// TIA Portal V18 export
FUNCTION "Block_LD" : Void   // FC2, LAD
{ S7_Optimized_Access := 'TRUE' }
// stored: SetENOAutomatically false
   VAR_TEMP
      "A" : Bool;
      "B" : Bool;
      C : Bool;
      D : Bool;
      QU : Bool;
      QD : Bool;
      PT : Time;
      ET : Time;
      PV : Int;
      CV : Int;
   END_VAR
BEGIN

REGION Network 1
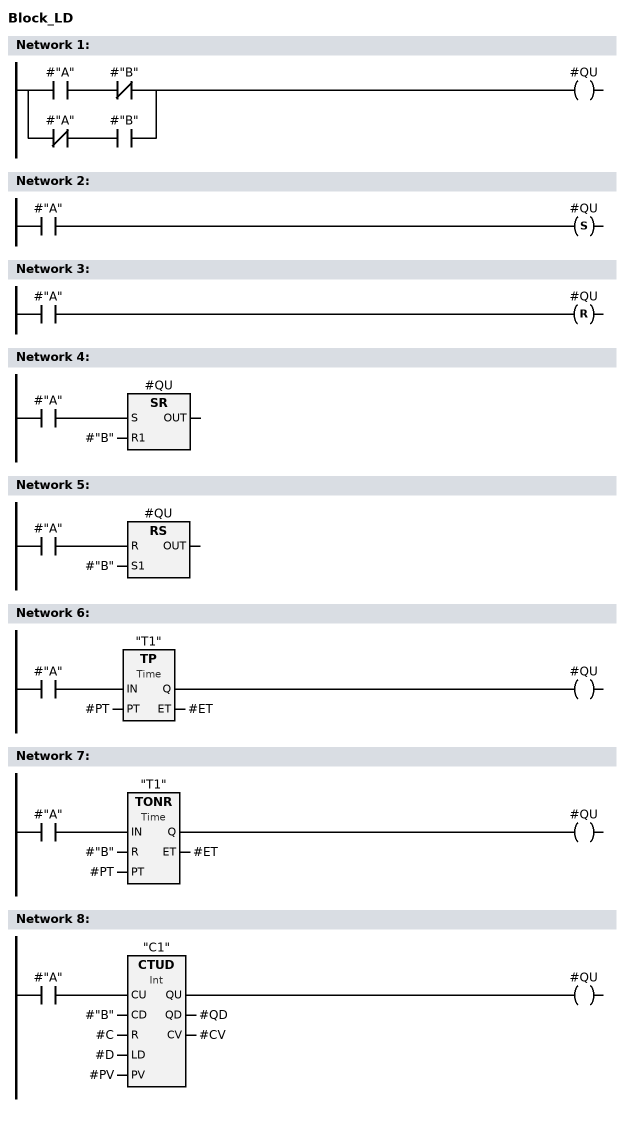
   RUNG wire#powerrail
      Contact( #"A" )
      I_Contact( #"B" )
      wire#w1
      Coil( #QU )
   END_RUNG
   RUNG wire#powerrail
      I_Contact( #"A" )
      Contact( #"B" )
   END_RUNG wire#w1
   // the same network as SCL:
   #QU := (#"A" AND NOT #"B") OR (NOT #"A" AND #"B");
END_REGION

REGION Network 2
   RUNG wire#powerrail
      Contact( #"A" )
      S_Coil( #QU )
   END_RUNG
   // the same network as SCL:
   IF #"A" THEN #QU := TRUE; END_IF;
END_REGION

REGION Network 3
   RUNG wire#powerrail
      Contact( #"A" )
      R_Coil( #QU )
   END_RUNG
   // the same network as SCL:
   IF #"A" THEN #QU := FALSE; END_IF;
END_REGION

REGION Network 4
   RUNG wire#powerrail
      Contact( #"A" )
      S_SR(operand := #QU, r1 := #"B")
   END_RUNG
   // the same network as SCL:
   IF #"A" THEN
       #QU := TRUE;   // SR flip-flop
   END_IF;
   IF #"B" THEN #QU := FALSE; END_IF;
END_REGION

REGION Network 5
   RUNG wire#powerrail
      Contact( #"A" )
      S_RS(operand := #QU, s1 := #"B")
   END_RUNG
   // the same network as SCL:
   IF #"A" THEN
       #QU := FALSE;   // RS flip-flop
   END_IF;
   IF #"B" THEN #QU := TRUE; END_IF;
END_REGION

REGION Network 6
   RUNG wire#powerrail
      Contact( #"A" )
      { S7_Templates := "time_type := Time" } "T1".TP(pt := #PT, et => #ET)
      Coil( #QU )
   END_RUNG
   // the same network as SCL:
   "T1".TP(IN := #"A", PT := #PT, ET => #ET);
   #QU := "T1".Q;
END_REGION

REGION Network 7
   RUNG wire#powerrail
      Contact( #"A" )
      { S7_Templates := "time_type := Time" } "T1".TONR(r := #"B", pt := #PT, et => #ET)
      Coil( #QU )
   END_RUNG
   // the same network as SCL:
   "T1".TONR(IN := #"A", R := #"B", PT := #PT, ET => #ET);
   #QU := "T1".Q;
END_REGION

REGION Network 8
   RUNG wire#powerrail
      Contact( #"A" )
      { S7_Templates := "value_type := Int" } "C1".CTUD(cd := #"B", r := #C, ld := #D, pv := #PV, qd => #QD, cv => #CV)
      Coil( #QU )
   END_RUNG
   // the same network as SCL:
   "C1".CTUD(CU := #"A", CD := #"B", R := #C, LD := #D, PV := #PV, QD => #QD, CV => #CV);
   #QU := "C1".QU;
END_REGION
END_FUNCTION
